FUNCTION_BLOCK ArrayCopier
  (* Standard: 61499-2 *)
  (* Version 0.1, 2016-00-15, Hammond, HAMMONDSDESKTOP *)
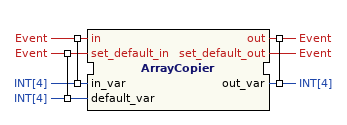
  EVENT_INPUT
    in WITH in_var;
    set_default_in WITH default_var;
  END_EVENT
  EVENT_OUTPUT
    out WITH out_var;
    set_default_out;
  END_EVENT
  VAR_INPUT
    in_var : ARRAY [0..3] OF INT;
    default_var : ARRAY [0..3] OF INT;
  END_VAR
  VAR_OUTPUT
    out_var : ARRAY [0..3] OF INT;
  END_VAR
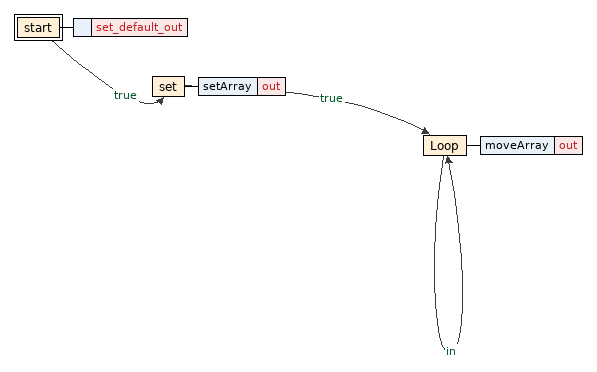
  EC_STATES
    start : -> set_default_out;
    set : setArray -> out;
    Loop : moveArray -> out;
  END_STATES
  EC_TRANSITIONS
    Loop TO Loop := in;
    set TO Loop := true;
    start TO set := true;
  END_TRANSITIONS
  ALGORITHM moveArray IN C:
me->out_var[0] = me->in_var[0];
me->out_var[1] = me->in_var[1];
me->out_var[2] = me->in_var[2];
me->out_var[3] = me->in_var[3];

printf("Set to %i %i %i %i\n", me->out_var[0], me->out_var[1], me->out_var[2], me->out_var[3]);
  END_ALGORITHM
  ALGORITHM setArray IN C:
me->out_var[0] = me->default_var[0];
me->out_var[1] = me->default_var[1];
me->out_var[2] = me->default_var[2];
me->out_var[3] = me->default_var[3];
  END_ALGORITHM
END_FUNCTION_BLOCK
